FUNCTION Array2D_Rows : UINT
VAR_IN_OUT CONSTANT
	A : ARRAY[*,*] OF LREAL;
END_VAR

IF UPPER_BOUND(A,1) < LOWER_BOUND(A,1) THEN
	Array2D_Rows := 0;
ELSE
	Array2D_Rows := DINT_TO_UINT(UPPER_BOUND(A,1) - LOWER_BOUND(A,1) + 1);
END_IF

END_FUNCTION

(* stored: Version 1.1.0.1, ProductVersion 3.1.4024.9
   POU Array2D_Rows: Id {62ad947c-b6a0-0ed8-1fe8-1b629cbe1f2f}, SpecialFunc None *)
